# EPICS StreamDevice protocol: protocols/xo.proto
Terminator = LF;
ExtraInput = Ignore;

setPlayloopLength {
	out "playloop_length %d";
	in;
}

getPlayloopLength {
	out "playloop_length";
	in "%d";
}

getPlayloopCursor {
	out "playloop_cursor";
	in "%d";
}

setAZ {
	out "dac20_autozero";
	wait 20000
	in "";
}
